FUNCTION_BLOCK Test_TStreamAdd_Read_UINT EXTENDS T_UnitTestBase
VAR
    Stream  : T_Stream(StreamLength := 2);
    ArgType : E_ArgTypeId := E_ArgTypeId.Type_UINT;
END_VAR

Stream.Init(2);

// add a UINT...
Stream.SetNextArgTypeId(ArgType);
Stream.Add_UINT(4567);

Stream.SetReadPosition(0);

// check next arg type is correct...
Assertion.AssertEquals_INT(Expected     := ArgType,
                           Actual       := Stream.GetNextArgTypeId(),
                           VariableName := 'Stream.GetNextArgTypeId()');

// check next value...	
Assertion.AssertEquals_UINT(Expected     := 4567,
                            Actual       := Stream.Read_UINT(),
                            VariableName := 'Stream.Read_UINT()');

// check we are at the end of the stream..							
Assertion.AssertEquals_UDINT(Expected     := Stream.StreamLength,
                             Actual       := Stream.ReadPosition,
                             VariableName := 'Stream.ReadPosition');

TestFinished();

END_FUNCTION_BLOCK

(* stored: Version 1.1.0.1, ProductVersion 3.1.4024.11
   POU Test_TStreamAdd_Read_UINT: Id {b902b738-8ad3-4380-b7ad-a8ed396d53ea}, SpecialFunc None *)
